{attribute 'qualified_only'}
VAR_GLOBAL
stParam : ST_Parameters;
stPlatform : ST_Platform;
END_VAR

(* stored: Version 1.1.0.1, ProductVersion 3.1.4024.12
   GVL G_Parameters: Id {669ea1f2-07fe-413d-92e6-ffdffa329b8e} *)
